# EPICS autosave request: ADFireWireWin/firewireWinApp/Db/firewireFeature_settings.req
$(P)$(R)$(FEATURE)
$(P)$(R)$(FEATURE)_CTRL
